TYPE ELL14KPolarisationFilterConfig EXTENDS DeviceConfiguration :
STRUCT
	SerialCommunication : SerialCommunication;
END_STRUCT
END_TYPE

(* stored: Version 1.1.0.1, ProductVersion 3.1.4024.4
   DUT ELL14KPolarisationFilterConfig: Id {d5672c2a-2727-4190-82df-e8d28c46e887} *)
